(* Schneider Machine Expert - Basic project limit switch, file version 2.7.0.0 *)
(* ProjectInformations: Name=New project *)

HARDWARE
  Cpu 0: TM200C24R
  EthernetConfiguration: NetworkName=M200, IpAllocationMode=FixedAddress, IpAddress=0.0.0.0, SubnetMask=0.0.0.0
  SerialLineConfiguration: Baud=Baud19200, Parity=ParityEven, DataBits=DataBits8, StopBits=StopBits1, PhysicalMedium=PhysicalMediumRs485, TransmissionMode=TransmissionModeModbusRtu, SlaveId=1, Addressing=SlaveAddressing
  MastTask: UsePeriodScanMode=false, PeriodScan=100
  FastTask: Period=255
  CpuBehavior: StartingMode=StartAsPreviousState, AutoSaveRamOnEeprom=true, WatchdogPeriod=250

SYMBOLS  (address, symbol, comment, settings)
  %M0         "mstop"
  %M4       MSTK3
  %I0.0       "start"
  %I0.1       "stop"
  %I0.2       "L1"
  %I0.3       "l2"
  %I0.4       "l3"
  %Q0.0       "k1"
  %Q0.1       "k2"
  %Q0.2       "k3"

POU New POU
  (* SectionNumber=1 *)

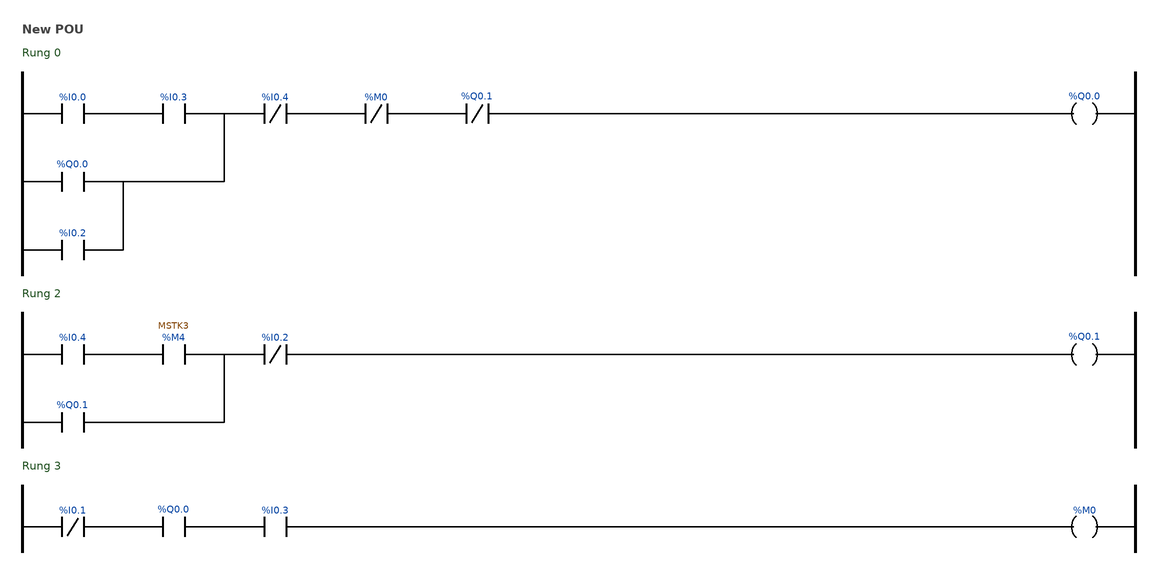

// Rung 0
  LD %I0.0
  AND %I0.3
  OR %Q0.0
  OR %I0.2
  ANDN %I0.4
  ANDN %M0
  ANDN %Q0.1
  ST %Q0.0
  // as ST:
  //   %Q0.0 := (%I0.0 AND %I0.3 OR %Q0.0 OR %I0.2) AND NOT %I0.4 AND NOT %M0 AND NOT %Q0.1;

// Rung 1
  LD %Q0.0
  OR %M4                  (* MSTK3 *)
  ANDN %Q0.1
  ST %M4                  (* MSTK3 *)
  // as ST:
  //   MSTK3 := (%Q0.0 OR MSTK3) AND NOT %Q0.1;
  (* the ladder stored for this rung does not match its IL; not drawn *)

// Rung 2
  LD %I0.4
  AND %M4                 (* MSTK3 *)
  OR %Q0.1
  ANDN %I0.2
  ST %Q0.1
  // as ST:
  //   %Q0.1 := (%I0.4 AND MSTK3 OR %Q0.1) AND NOT %I0.2;

// Rung 3
  LDN %I0.1
  AND %Q0.0
  AND %I0.3
  ST %M0
  // as ST:
  //   %M0 := NOT %I0.1 AND %Q0.0 AND %I0.3;
